TYPE ST_ergonomicCtrlData :
STRUCT
	m_monitorHeight : LREAL;
	m_headAngle : LREAL;
	m_handrailHeight : LREAL;
	m_footDistance : LREAL;
END_STRUCT
END_TYPE

(* stored: Version 1.1.0.1, ProductVersion 3.1.4024.11
   DUT ST_ergonomicCtrlData: Id {476619f7-fa03-4b2e-ad16-ef2a94d0f41f} *)
